# EPICS StreamDevice protocol: apps/srsApp/Db/srs-rga.proto
#
# N. Baltzell, 2022
#
# EPICS support for Stanford Research Systems RGA-X00
#
# Adapted from John Sinclair, sincalairjw@ornl.gov, 2/18/2015
#

OutTerminator = "\r\n";
InTerminator = "\n\r";
ExtraInput = Ignore;

command   { out "\$1"; }
getString { out "\$1?"; in "%s"; }
getInt    { out "\$1?"; in "%d"; }
getFloat  { out "\$1?"; in "%f"; }
putFloat  { out "\$1 %f"; }
putInt    { out "\$1 %d"; }

scan {
    ReplyTimeout = 30000;
    ReadTimeout = 30000;
    InTerminator =;
    out "\$1 1";
    in "%#4r%*r";
}

mass {
    ReplyTimeout = 3000;
    ReadTimeout = 3000;
    InTerminator = ;
    out "MR%(\$1.VAL)d";
    in  "%#4r";
}
